FUNCTION_BLOCK FB_LamparaConmutada_LD_2
// La lampara se enciende si estando apagada se acciona el pulsador
// La lampara se apaga si estando encendida se acciona el pulsador
VAR
    Pulsacion         : R_TRIG;
    MemoriaLampara    : BOOL;
    Lampara   AT %Q*  : BOOL;
    Pulsador  AT %I*  : BOOL;
END_VAR

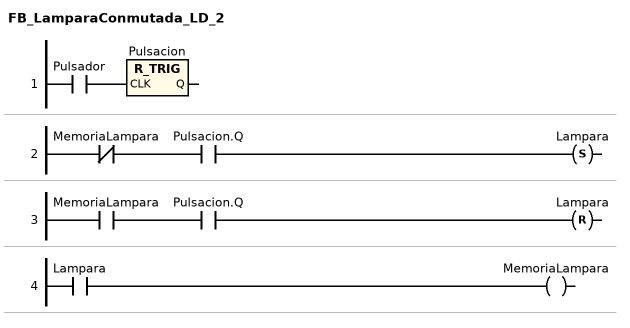
// NETWORK 1
Pulsacion(CLK := Pulsador); // R_TRIG

// NETWORK 2
Lampara S= NOT MemoriaLampara AND Pulsacion.Q;

// NETWORK 3
Lampara R= MemoriaLampara AND Pulsacion.Q;

// NETWORK 4
MemoriaLampara := Lampara;

END_FUNCTION_BLOCK

(* stored: Version 1.1.0.1, ProductVersion 3.1.4024.15
   POU FB_LamparaConmutada_LD_2: Id {d6c70e8d-eab6-4aa2-8559-701d0e77a92e}, SpecialFunc None *)
